// Mitsubishi GX Works2 project: IELET2103_Datalab7   PLC: FX2N/FX2NC
// IELET2103_Datalab7.gxw

// global labels: Global1
VAR_GLOBAL
  Stopp AT X000 : BOOL;
  Start AT X001 : BOOL;
  EndestillingA AT X002 : BOOL;
  EndestillingC AT X003 : BOOL;
  MidtstillingB AT X004 : BOOL;
  Nødstopp AT X005 : BOOL;
  Feil_i_anlegget AT X006 : BOOL;
  KvitteringAvAlarm AT X007 : BOOL;
  VognFrem AT Y000 : BOOL;
  VognTilbake AT Y001 : BOOL;
  MagnetventilForAapningAvSpjeld AT Y002 : BOOL;
  MagnetventilForLukkingAvSpjeld AT Y003 : BOOL;
END_VAR

// task Task_01 (event TRUE, interval 0, priority 31): Oppgave1a)

PROGRAM Oppgave1a)
(* structured ladder/FBD written out as ST: instructions are called as NAME(EN, inputs, outputs); _pN, _eN, _tN stand for wires *)
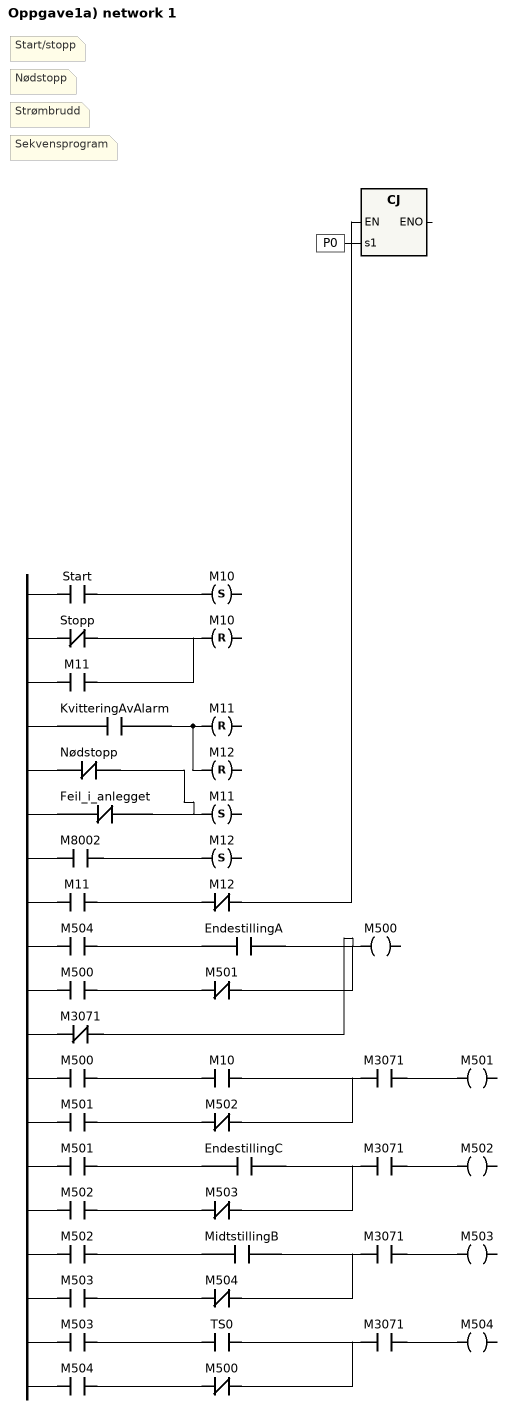
(* network 1 *)
(* Start/stopp *)
(* Nødstopp *)
(* Strømbrudd *)
(* Sekvensprogram *)
SET(Start, M10);
RST((NOT Stopp) OR M11, M10);
RST(KvitteringAvAlarm, M11);
RST(KvitteringAvAlarm, M12);
SET((NOT Nødstopp) OR (NOT Feil_i_anlegget), M11);
SET(M8002, M12);
CJ(M11 AND NOT M12, P0);
M500 := (M504 AND EndestillingA) OR (M500 AND NOT M501) OR (NOT M3071);
M501 := ((M500 AND M10) OR (M501 AND NOT M502)) AND M3071;
M502 := ((M501 AND EndestillingC) OR (M502 AND NOT M503)) AND M3071;
M503 := ((M502 AND MidtstillingB) OR (M503 AND NOT M504)) AND M3071;
M504 := ((M503 AND TS0) OR (M504 AND NOT M500)) AND M3071;
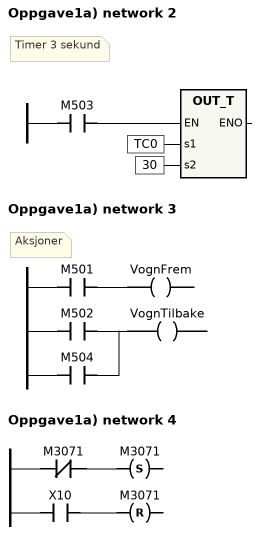
(* network 2 P0: *)
(* Timer 3 sekund *)
OUT_T(M503, TC0, 30);
(* network 3 *)
(* Aksjoner *)
VognFrem := M501;
VognTilbake := M502 OR M504;
(* network 4 *)
SET(NOT M3071, M3071);
RST(X10, M3071);
END_PROGRAM
